FUNCTION_BLOCK "LAnyAxis_MC_TorqueLimiting"
{ S7_Optimized_Access := 'TRUE' }
AUTHOR : 'tech.team.motioncontrol@siemens.com'
FAMILY : AnyAxis
VERSION : 1.0
   VAR_INPUT
      Axis : DB_ANY;
      Enable : Bool;
      Limit : LReal := -1.0;
      Mode : DInt;
   END_VAR

   VAR_OUTPUT
      InClamping { ExternalWritable := 'False'} : Bool;
      InLimitation { ExternalWritable := 'False'} : Bool;
      Busy { ExternalWritable := 'False'} : Bool;
      Error { ExternalWritable := 'False'} : Bool;
      ErrorId { ExternalWritable := 'False'} : Word;
   END_VAR

   VAR
      instMC {InstructionName := 'MC_TORQUELIMITING'; LibVersion := '6.0'; ExternalAccessible := 'False'; ExternalVisible := 'False'; ExternalWritable := 'False'; S7_SetPoint := 'False'} : MC_TORQUELIMITING;
      statEnableOld { ExternalAccessible := 'False'; ExternalVisible := 'False'; ExternalWritable := 'False'} : Bool;
      statAxis { ExternalAccessible := 'False'; ExternalVisible := 'False'; ExternalWritable := 'False'} : DB_ANY;
      statAxisType { ExternalAccessible := 'False'; ExternalVisible := 'False'; ExternalWritable := 'False'} : Int;
   END_VAR

   VAR CONSTANT
      ERROR_INVALID_TECHNOLOGY_OBJECT : Word := 16#8002;
      IDLE : Int := 0;
      INVALID_AXIS : Int := -1;
      SPEED_AXIS : Int := 2;
      POSITIONING_AXIS : Int := 3;
      SYNCHRONOUS_AXIS : Int := 4;
   END_VAR


BEGIN
	REGION HEADER
	    //================================================================================
	    // SIEMENS AG
	    // (c)Copyright 2020 All Rights Reserved
	    //--------------------------------------------------------------------------------
	    // Library: LAnyAxis
	    // Tested with: S7-1515-2 PN
	    // Engineering: TIA Portal V16
	    // Restrictions: -
	    // Requirements: S7-1500 FW 2.8.1
	    // Functionality: Conversion DB_ANY --> TO_Axis
	    // Support: tech.team.motioncontrol@siemens.com
	    // Note: Parameter comments are only available in language 'English (United States)'
	    //--------------------------------------------------------------------------------
	    // Change log table:
	    // Version  Date        Expert in charge  Changes applied
	    // 01.00.00 10.03.2020  RS                First released version
	    //================================================================================
	END_REGION

	REGION ENABLE
	    IF (#statAxisType = #IDLE) AND #Enable THEN
	        // Check axis type
	        CASE TypeOfDB(#Axis) OF
	            TO_POSITIONINGAXIS:
	                #statAxisType := #POSITIONING_AXIS;
	                #statAxis := #Axis;

	            TO_SYNCHRONOUSAXIS:
	                #statAxisType := #SYNCHRONOUS_AXIS;
	                #statAxis := #Axis;

	            TO_SPEEDAXIS:
	                #statAxisType := #SPEED_AXIS;
	                #statAxis := #Axis;

	            ELSE
	                #statAxisType := #INVALID_AXIS;
	                #statAxis := 0;
	        END_CASE;

	    ELSIF NOT #Enable AND (#statAxisType = #INVALID_AXIS) THEN
	        #statAxisType := #IDLE;

	        // Outputs
	        #InClamping := FALSE;
	        #InLimitation := FALSE;
	        #Busy := FALSE;
	        #Error := FALSE;
	        #ErrorId := 16#0;
	    END_IF;

	    // Edge detection
	    #statEnableOld := #Enable;
	END_REGION

	CASE #statAxisType OF
	    #IDLE:
	        ;

	    #POSITIONING_AXIS,
	    #SYNCHRONOUS_AXIS,
	    #SPEED_AXIS:
	        REGION VALID_AXIS
	            // Inputs
	            #instMC.Enable := #Enable;
	            #instMC.Limit := #Limit;
	            #instMC.Mode := #Mode;

	            // Call of MC instruction
	            CASE #statAxisType OF
	                #POSITIONING_AXIS:
	                    "LAnyAxis_UnpubTorqueLimitingPosAxis"(axis := #statAxis,
	                                                          instMC := #instMC);
	                #SYNCHRONOUS_AXIS:
	                    "LAnyAxis_UnpubTorqueLimitingSyncAxis"(axis := #statAxis,
	                                                           instMC := #instMC);
	                #SPEED_AXIS:
	                    "LAnyAxis_UnpubTorqueLimitingSpeedAxis"(axis := #statAxis,
	                                                            instMC := #instMC);
	            END_CASE;

	            // Outputs
	            #InClamping := #instMC.InClamping;
	            #InLimitation := #instMC.InLimitation;
	            #Busy := #instMC.Busy;
	            #Error := #instMC.Error;
	            #ErrorId := #instMC.ErrorId;

	            // Status of MC instruction
	            IF NOT #instMC.Busy
	                AND NOT #instMC.Error
	            THEN
	                // Not active
	                #statAxisType := #IDLE;
	            END_IF;
	        END_REGION

	    ELSE
	        REGION INVALID_AXIS
	            // Outputs
	            #InClamping := FALSE;
	            #InLimitation := FALSE;
	            #Busy := FALSE;
	            #Error := TRUE;
	            #ErrorId := #ERROR_INVALID_TECHNOLOGY_OBJECT;
	        END_REGION
	END_CASE;
END_FUNCTION_BLOCK

